KUKA KRL program: wkz1_ab.src, wkz1_ab.dat

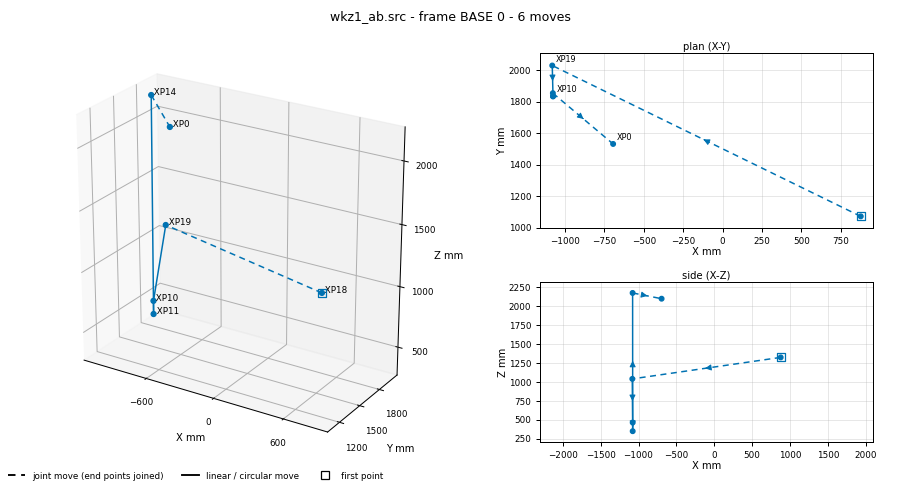
[picture p0: tool path of wkz1_ab.src in frame BASE 0, 6 of 6 moves have a stored position in this frame; points joined in program order, loops and branches not executed]
--- wkz1_ab.src ---
&ACCESS RVO3
&REL 1
&COMMENT Deposita Pinca C1
&PARAM DISKPATH = KRC:\R1\Program
&PARAM TEMPLATE = C:\KRC\Roboter\Template\vorgabe
&PARAM EDITMASK = *
DEF wkz1_ab( )
;FOLD INI
  ;FOLD BASISTECH INI
    GLOBAL INTERRUPT DECL 3 WHEN $STOPMESS==TRUE DO IR_STOPM ( )
    INTERRUPT ON 3
    BAS (#INITMOV,0 )
  ;ENDFOLD (BASISTECH INI)
;FOLD GRIPPERTECH INI
USER_GRP(0,DUMMY,DUMMY,GDEFAULT)
;ENDFOLD (GRIPPERTECH INI)
  ;FOLD USER INI
    ;Make your modifications here

  ;ENDFOLD (USER INI)
;ENDFOLD (INI);FOLD ;%{PE}%R 8.2.20,%MKUKATPBASIS,%CCOMMENT,%VNORMAL,%P 2:

; Caracterização dos meios de produção:
; Versão Atual:
; 15/07/2013 12:00 Name: P13.050-R4 CHANGES: Deposita Pinça
; C1


chk_w1_wechs_ok ( )     ; CHECK FERRAMENTA: C1


;FOLD PTP P18 CONT Vel=100 % PDAT9 Tool[8]:TOOL_CHANGE Base[0];%{PE}%R 8.2.20,%MKUKATPBASIS,%CMOVE,%VPTP,%P 1:PTP, 2:P18, 3:C_DIS, 5:100, 7:PDAT9
$BWDSTART=FALSE
PDAT_ACT=PPDAT9
FDAT_ACT=FP18
BAS(#PTP_PARAMS,100)
PTP XP18 C_DIS
;ENDFOLD

;FOLD PULSE 183 'DOCK 3 Abrir Proteção' State=TRUE CONT Time=1 sec;%{PE}%R 8.2.20,%MKUKATPBASIS,%COUT,%VPULSE,%P 2:183, 3:DOCK 3 Abrir Proteção, 5:TRUE, 6:CONTINUE, 8:1
CONTINUE
PULSE($OUT[183], TRUE,1)
;ENDFOLD
;FOLD WAIT FOR ( IN 219 'Posicao p/ Acoplamento OK' ) CONT;%{PE}%R 8.2.20,%MKUKATPBASIS,%CEXT_WAIT_FOR,%VEXT_WAIT_FOR,%P 2:, 4:, 5:$IN, 6:219, 7:Posicao p/ Acoplamento OK, 9:CONTINUE
CONTINUE
WAIT FOR  ( $IN[219] )
;ENDFOLD
;FOLD WAIT FOR NOT ( IN 177 'DOCK 3 Deposito Ocupado' ) CONT;%{PE}%R 8.2.20,%MKUKATPBASIS,%CEXT_WAIT_FOR,%VEXT_WAIT_FOR,%P 2:NOT, 4:, 5:$IN, 6:177, 7:DOCK 3 Deposito Ocupado, 9:CONTINUE
CONTINUE
WAIT FOR  NOT ( $IN[177] )
;ENDFOLD
;FOLD WAIT FOR ( IN 181 'DOCK 3 Proteção Aberta' ) CONT;%{PE}%R 8.2.20,%MKUKATPBASIS,%CEXT_WAIT_FOR,%VEXT_WAIT_FOR,%P 2:, 4:, 5:$IN, 6:181, 7:DOCK 3 Proteção Aberta, 9:CONTINUE
CONTINUE
WAIT FOR  ( $IN[181] )
;ENDFOLD
;FOLD WAIT FOR NOT ( IN 182 'DOCK 3 Proteção Fechada' ) CONT;%{PE}%R 8.2.20,%MKUKATPBASIS,%CEXT_WAIT_FOR,%VEXT_WAIT_FOR,%P 2:NOT, 4:, 5:$IN, 6:182, 7:DOCK 3 Proteção Fechada, 9:CONTINUE
CONTINUE
WAIT FOR  NOT ( $IN[182] )
;ENDFOLD

;FOLD PTP P19 CONT Vel=100 % PDAT10 Tool[8]:TOOL_CHANGE Base[0];%{PE}%R 8.2.20,%MKUKATPBASIS,%CMOVE,%VPTP,%P 1:PTP, 2:P19, 3:C_DIS, 5:100, 7:PDAT10
$BWDSTART=FALSE
PDAT_ACT=PPDAT10
FDAT_ACT=FP19
BAS(#PTP_PARAMS,100)
PTP XP19 C_DIS
;ENDFOLD

;FOLD LIN P10 CONT Vel=1 m/s CPDAT5 Tool[8]:TOOL_CHANGE Base[0];%{PE}%R 8.2.20,%MKUKATPBASIS,%CMOVE,%VLIN,%P 1:LIN, 2:P10, 3:C_DIS C_DIS, 5:1, 7:CPDAT5
$BWDSTART=FALSE
LDAT_ACT=LCPDAT5
FDAT_ACT=FP10
BAS(#CP_PARAMS,1)
LIN XP10 C_DIS C_DIS
;ENDFOLD

;FOLD ; PONTO DE DEPOSITO DA PINCA;%{PE}%R 8.2.19,%MKUKATPBASIS,%CCOMMENT,%VNORMAL,%P 2:PONTO  DE  DEPOSITO  DA  PINCA
;ENDFOLD
;FOLD LIN P11 Vel=0.1 m/s CPDAT6 Tool[1]:GUN_C1 Base[0];%{PE}%R 8.2.20,%MKUKATPBASIS,%CMOVE,%VLIN,%P 1:LIN, 2:P11, 3:, 5:0.1, 7:CPDAT6
$BWDSTART=FALSE
LDAT_ACT=LCPDAT6
FDAT_ACT=FP11
BAS(#CP_PARAMS,0.1)
LIN XP11
;ENDFOLD
;FOLD  ;%{PE}%R 8.2.19,%MKUKATPBASIS,%CCOMMENT,%VNORMAL,%P 2:
;ENDFOLD
;FOLD WAIT FOR ( IN 222 'Liberacao p/ Desbloqueio' );%{PE}%R 8.2.20,%MKUKATPBASIS,%CEXT_WAIT_FOR,%VEXT_WAIT_FOR,%P 2:, 4:, 5:$IN, 6:222, 7:Liberacao p/ Desbloqueio, 9:
WAIT FOR  ( $IN[222] )
;ENDFOLD
;FOLD WAIT FOR ( IN 177 'DOCK 3 Deposito Ocupado' );%{PE}%R 8.2.20,%MKUKATPBASIS,%CEXT_WAIT_FOR,%VEXT_WAIT_FOR,%P 2:, 4:, 5:$IN, 6:177, 7:DOCK 3 Deposito Ocupado, 9:
WAIT FOR  ( $IN[177] )
;ENDFOLD
;FOLD WAIT Time=0.3 sec;%{PE}%R 8.2.20,%MKUKATPBASIS,%CWAIT,%VWAIT,%P 3:0.3
WAIT SEC 0.3
;ENDFOLD
;FOLD OUT 224 'Bloquear MPS' State=FALSE ;%{PE}%R 8.2.20,%MKUKATPBASIS,%COUT,%VOUTX,%P 2:224, 3:Bloquear MPS, 5:FALSE, 6:
$OUT[224]=FALSE
;ENDFOLD
;FOLD OUT 223 'Desbloquear MPS' State=TRUE ;%{PE}%R 8.2.20,%MKUKATPBASIS,%COUT,%VOUTX,%P 2:223, 3:Desbloquear MPS, 5:TRUE, 6:
$OUT[223]=TRUE
;ENDFOLD
;FOLD WAIT FOR ( IN 217 'MPS Destravado' );%{PE}%R 8.2.20,%MKUKATPBASIS,%CEXT_WAIT_FOR,%VEXT_WAIT_FOR,%P 2:, 4:, 5:$IN, 6:217, 7:MPS Destravado, 9:
WAIT FOR  ( $IN[217] )
;ENDFOLD
;FOLD WAIT FOR NOT ( IN 221 'MPS Travado' );%{PE}%R 8.2.20,%MKUKATPBASIS,%CEXT_WAIT_FOR,%VEXT_WAIT_FOR,%P 2:NOT, 4:, 5:$IN, 6:221, 7:MPS Travado, 9:
WAIT FOR  NOT ( $IN[221] )
;ENDFOLD
;FOLD IBUS OFF;%{PE}%R 8.2.20,%MKUKATPBASIS,%CIBUS,%VMAP,%P 2:#OFF, 3:1
$IBUS_OFF=$IBUS_ON
$IBUS_ON=0
;ENDFOLD
;FOLD WAIT Time=0.2 sec;%{PE}%R 8.2.20,%MKUKATPBASIS,%CWAIT,%VWAIT,%P 3:0.2
WAIT SEC 0.2
;ENDFOLD

;FOLD LIN P14 Vel=0.5 m/s CPDAT9 Tool[8]:TOOL_CHANGE Base[0];%{PE}%R 8.2.20,%MKUKATPBASIS,%CMOVE,%VLIN,%P 1:LIN, 2:P14, 3:, 5:0.5, 7:CPDAT9
$BWDSTART=FALSE
LDAT_ACT=LCPDAT9
FDAT_ACT=FP14
BAS(#CP_PARAMS,0.5)
LIN XP14
;ENDFOLD

;FOLD WAIT FOR ( IN 177 'DOCK 3 Deposito Ocupado' ) CONT;%{PE}%R 8.2.20,%MKUKATPBASIS,%CEXT_WAIT_FOR,%VEXT_WAIT_FOR,%P 2:, 4:, 5:$IN, 6:177, 7:DOCK 3 Deposito Ocupado, 9:CONTINUE
CONTINUE
WAIT FOR  ( $IN[177] )
;ENDFOLD
;FOLD WAIT FOR NOT ( IN 219 'Posicao p/ Acoplamento OK' ) CONT;%{PE}%R 8.2.20,%MKUKATPBASIS,%CEXT_WAIT_FOR,%VEXT_WAIT_FOR,%P 2:NOT, 4:, 5:$IN, 6:219, 7:Posicao p/ Acoplamento OK, 9:CONTINUE
CONTINUE
WAIT FOR  NOT ( $IN[219] )
;ENDFOLD
;FOLD OUT 223 'Desbloquear MPS' State=FALSE CONT;%{PE}%R 8.2.20,%MKUKATPBASIS,%COUT,%VOUTX,%P 2:223, 3:Desbloquear MPS, 5:FALSE, 6:CONTINUE
CONTINUE
$OUT[223]=FALSE
;ENDFOLD

;FOLD PTP P0 CONT Vel=100 % PDAT0 Tool[8]:TOOL_CHANGE Base[0];%{PE}%R 8.2.20,%MKUKATPBASIS,%CMOVE,%VPTP,%P 1:PTP, 2:P0, 3:C_DIS, 5:100, 7:PDAT0
$BWDSTART=FALSE
PDAT_ACT=PPDAT0
FDAT_ACT=FP0
BAS(#PTP_PARAMS,100)
PTP XP0 C_DIS
;ENDFOLD

;FOLD PULSE 184 'DOCK 3 Fechar Proteção' State=TRUE Time=1 sec;%{PE}%R 8.2.20,%MKUKATPBASIS,%COUT,%VPULSE,%P 2:184, 3:DOCK 3 Fechar Proteção, 5:TRUE, 6:, 8:1
PULSE($OUT[184], TRUE,1)
;ENDFOLD

END

--- wkz1_ab.dat ---
&ACCESS RVO3
&REL 1
&COMMENT Deposita Pinca C1
&PARAM DISKPATH = KRC:\R1\Program
&PARAM TEMPLATE = C:\KRC\Roboter\Template\vorgabe
&PARAM EDITMASK = *
DEFDAT wkz1_ab
;FOLD EXTERNAL DECLARATIONS;%{PE}%MKUKATPBASIS,%CEXT,%VCOMMON,%P
;FOLD GRIPPERTECH EXT
EXT  H50 (INT  :IN,INT  :IN,INT  :IN,GRP_TYP  :IN )
;ENDFOLD (GRIPPERTECH EXT)
;FOLD SPOTTECH EXT
EXT  USERSPOT (S_COMMAND  :IN,SPOT_TYPE  :IN )
;ENDFOLD (SPOTTECH EXT)
;FOLD BASISTECH EXT;%{PE}%MKUKATPBASIS,%CEXT,%VEXT,%P
EXT  BAS (BAS_COMMAND  :IN,REAL  :IN )
DECL INT SUCCESS
;ENDFOLD (BASISTECH EXT)
;FOLD USER EXT;%{E}%MKUKATPUSER,%CEXT,%VEXT,%P
;Make your modifications here

;ENDFOLD (USER EXT)
;ENDFOLD (EXTERNAL DECLARATIONS)
DECL BASIS_SUGG_T LAST_BASIS={POINT1[] "P0                      ",POINT2[] "P0                      ",CP_PARAMS[] "CPDAT0                  ",PTP_PARAMS[] "PDAT0                   ",CONT[] "                        ",CP_VEL[] "0.5                     ",PTP_VEL[] " 100                    ",SYNC_PARAMS[] "SYNCDAT                 ",SPL_NAME[] "S0                      "}
DECL PDAT PPDAT0={VEL 100.0,ACC 100.0,APO_DIST 100.0,APO_MODE #CDIS}
DECL E6POS XP0={X -695.183899,Y 1533.36206,Z 2101.271,A -87.8347015,B -0.405478299,C 176.795898,S 2,T 43,E1 -47.1511002,E2 0.0,E3 0.0,E4 0.0,E5 0.0,E6 0.0}
DECL FDAT FP0={TOOL_NO 8,BASE_NO 0,IPO_FRAME #BASE,POINT2[] " ",TQ_STATE FALSE}
DECL LDAT LCPDAT5={VEL 2.0,ACC 100.0,APO_DIST 100.0,APO_FAC 50.0,AXIS_VEL 100.0,AXIS_ACC 100.0,ORI_TYP #VAR,CIRC_TYP #BASE,JERK_FAC 50.0,GEAR_JERK 50.0,EXAX_IGN 0}
DECL E6POS XP10={X -1076.89099,Y 1836.65295,Z 465.5849,A -89.1070786,B -0.753481805,C -0.0323741809,S 2,T 43,E1 -351.006104,E2 0.0,E3 0.0,E4 0.0,E5 0.0,E6 0.0}
DECL FDAT FP10={TOOL_NO 1,BASE_NO 0,IPO_FRAME #BASE,POINT2[] " ",TQ_STATE FALSE}
DECL LDAT LCPDAT6={VEL 2.0,ACC 100.0,APO_DIST 100.0,APO_FAC 50.0,AXIS_VEL 100.0,AXIS_ACC 100.0,ORI_TYP #VAR,CIRC_TYP #BASE,JERK_FAC 50.0,GEAR_JERK 50.0,EXAX_IGN 0}
DECL E6POS XP11={X -1076.93201,Y 1835.14795,Z 351.299011,A -89.1070633,B -0.753454983,C -0.0324217007,S 2,T 43,E1 -351.006287,E2 0.0,E3 0.0,E4 0.0,E5 0.0,E6 0.0}
DECL FDAT FP11={TOOL_NO 1,BASE_NO 0,IPO_FRAME #BASE,POINT2[] " ",TQ_STATE FALSE}
DECL E6POS XP14={X -1077.91394,Y 1856.05005,Z 2177.354,A -74.3145218,B 0.1208717,C 179.640106,S 2,T 43,E1 -351.014893,E2 0.0,E3 0.0,E4 0.0,E5 0.0,E6 0.0}
DECL FDAT FP14={TOOL_NO 8,BASE_NO 0,IPO_FRAME #BASE,POINT2[] " ",TQ_STATE FALSE}
DECL LDAT LCPDAT9={VEL 2.0,ACC 100.0,APO_DIST 100.0,APO_FAC 50.0,AXIS_VEL 100.0,AXIS_ACC 100.0,ORI_TYP #VAR,CIRC_TYP #BASE,JERK_FAC 50.0,GEAR_JERK 50.0,EXAX_IGN 0}
DECL PDAT PPDAT9={VEL 100.0,ACC 100.0,APO_DIST 100.0,APO_MODE #CDIS}
DECL E6POS XP18={X 877.703918,Y 1073.51196,Z 1325.97498,A -136.596893,B 8.38269615,C 4.37436914,S 2,T 3,E1 -351.040894,E2 0.0,E3 0.0,E4 0.0,E5 0.0,E6 0.0}
DECL FDAT FP18={TOOL_NO 1,BASE_NO 0,IPO_FRAME #BASE,POINT2[] " ",TQ_STATE FALSE}
DECL PDAT PPDAT10={VEL 100.0,ACC 100.0,APO_DIST 100.0,APO_MODE #CDIS}
DECL E6POS XP19={X -1081.77502,Y 2031.49695,Z 1042.354,A -89.902771,B 1.26391304,C -0.392126113,S 2,T 35,E1 -351.021393,E2 0.0,E3 0.0,E4 0.0,E5 0.0,E6 0.0}
DECL FDAT FP19={TOOL_NO 1,BASE_NO 0,IPO_FRAME #BASE,POINT2[] " ",TQ_STATE FALSE}
ENDDAT
